screen "HAND_3" 800x480
   Button "Button_2" at 5,415 size 191x62; TextOff 'BACK'
      on Click: ActivateScreen("HAND_2", 0)
   TextField "Text field_12" at 206,35 size 347x29; Text 'CONVEYOR -1 START/STOP'
   Button "Button_21" at 690,7 size 11x44; TextOff 'Text'; PictureOff "Untitled_2"
   Button "Button_22" at 703,7 size 65x94; TextOff 'Text'; PictureOn "RIGHT_ARROW_ACTIVE"; PictureOff "RIGHT_ARROW_1"
      on Press: function_b14e0dd5("CONVEYOR -1 RUN FROM HMI", 0)
   TextField "Text field_13" at 623,7 size 64x44; Text 'START'
   TextField "Text field_18" at 623,57 size 64x44; Text 'Q1.0'
      Appearance <- "Tag_12"
   Button "Button_23" at 690,57 size 11x44; TextOff 'Text'; PictureOff "Untitled_2"
   Button "Button_24" at 33,7 size 65x94; TextOff 'Text'; PictureOn "LEFT_ARROW_ACTIVE"; PictureOff "LEFT_ARR"
      on Press: function_b14e0dd5("CONVEYOR -1 STOP FROM HMI", 0)
   TextField "Text field_19" at 119,7 size 64x44; Text 'STOP'
   Button "Button_25" at 101,7 size 11x44; TextOff 'Text'; PictureOff "Untitled_2"
   TextField "Text field_20" at 119,57 size 64x44; Text 'Q1.0'
      Appearance <- "Tag_12"
   Button "Button_26" at 101,57 size 11x44; TextOff 'Text'; PictureOff "Untitled_2"
   TextField "Text field_5" at 207,134 size 347x29; Text 'CONVEYOR -2 START/STOP'
   Button "Button_3" at 691,106 size 11x44; TextOff 'Text'; PictureOff "Untitled_2"
   Button "Button_4" at 704,106 size 65x94; TextOff 'Text'; PictureOn "RIGHT_ARROW_ACTIVE"; PictureOff "RIGHT_ARROW_1"
      on Press: function_b14e0dd5("CONVEYOR 2 RUN FROM HMI", 0)
   TextField "Text field_6" at 624,106 size 64x44; Text 'START'
   TextField "Text field_7" at 624,156 size 64x44; Text 'Q1.1'
      Appearance <- "Tag_13"
   Button "Button_5" at 691,156 size 11x44; TextOff 'Text'; PictureOff "Untitled_2"
   Button "Button_6" at 34,106 size 65x94; TextOff 'Text'; PictureOn "LEFT_ARROW_ACTIVE"; PictureOff "LEFT_ARR"
      on Press: function_b14e0dd5("CONVEYOR -2 STOP FROM HMI", 0)
   TextField "Text field_8" at 120,106 size 64x44; Text 'STOP'
   Button "Button_7" at 102,106 size 11x44; TextOff 'Text'; PictureOff "Untitled_2"
   TextField "Text field_9" at 120,156 size 64x44; Text 'Q1.1'
      Appearance <- "Tag_13"
   Button "Button_8" at 102,156 size 11x44; TextOff 'Text'; PictureOff "Untitled_2"
   TextField "Text field_1" at 236,241 size 327x29; Text 'PLUG HOLDER HOLD/UNHOLD'
   Button "Button_9" at 690,213 size 11x44; TextOff 'Text'; PictureOff "Untitled_2"
   Button "Button_10" at 703,213 size 65x94; TextOff 'Text'; PictureOn "RIGHT_ARROW_ACTIVE"; PictureOff "RIGHT_ARROW_1"
      on Press: function_b14e0dd5("HMI_GRIPPER_HOLD", 0)
      Appearance <- "HMI_GRIPPER_HOLD"
   TextField "Text field_2" at 623,213 size 64x44; Text 'HOLD'
      Appearance <- "GRIPPER_HOLD"
   TextField "Text field_3" at 623,263 size 64x44; Text 'Q6.2'
      Appearance <- "GRIPPER_HOLD"
   Button "Button_11" at 690,263 size 11x44; TextOff 'Text'; PictureOff "Untitled_2"
   Button "Button_12" at 33,213 size 65x94; TextOff 'Text'; PictureOn "LEFT_ARROW_ACTIVE"; PictureOff "LEFT_ARR"
      on Press: function_b14e0dd5("HMI_GRIPPER_UNHOLD", 0)
      Appearance <- "HMI_GRIPPER_UNHOLD"
   TextField "Text field_4" at 119,213 size 64x44; Text 'UNHOLD'
      Appearance <- "GRIPPER_UNHOLD"
   Button "Button_13" at 101,213 size 11x44; TextOff 'Text'; PictureOff "Untitled_2"
   TextField "Text field_10" at 119,263 size 64x44; Text 'Q6.3'
      Appearance <- "GRIPPER_UNHOLD"
   Button "Button_14" at 101,263 size 11x44; TextOff 'Text'; PictureOff "Untitled_2"
   Button "Button_27" at 609,416 size 191x63; TextOff 'HOME'
      on Click: ActivateScreen("MAIN", 0)
   Softkey "Softkey_F1" at 0,0 size 0x0
      on KeyDown: ActivateScreen("HAND_2", 0)
   Softkey "Softkey_F8" at 0,0 size 0x0
      on KeyDown: ActivateScreen("MAIN", 0)

screen "INPUT LIST" 800x480
   SymbolicIOField "Symbolic I/O field_1" at 160,52 size 153x48; TextOn '1'; TextOff '0'; TextList "INPUT ADDRESS"
      ProcessValue <- "0_BIT"
   SymbolicIOField "Symbolic I/O field_2" at 315,52 size 474x48; TextOn '1'; TextOff '0'; TextList "INPUT ADDRESS COMMENT"
      ProcessValue <- "0_BIT"
   TextField "Text field_1" at 36,14 size 71x23; Text 'STATUS'
   TextField "Text field_2" at 188,13 size 68x23; Text 'INPUTS'
   TextField "Text field_3" at 350,13 size 99x23; Text 'COMMENTS'
   SymbolicIOField "Symbolic I/O field_3" at 620,3 size 167x48; TextOn '1'; TextOff '0'; TextList "INPUT BYTE SELECTION"
      on Activate: function_dbe01993("0_BIT", 8, "BYTE SELECTION", 0); function_dbe01993("1_BIT", 8, "BYTE SELECTION", 1); function_dbe01993("2_BIT", 8, "BYTE SELECTION", 2); function_dbe01993("3_BIT", 8, "BYTE SELECTION", 3); function_dbe01993("4_BIT", 8, "BYTE SELECTION", 4); function_dbe01993("5_BIT", 8, "BYTE SELECTION", 5); function_dbe01993("6_BIT", 8, "BYTE SELECTION", 6); function_dbe01993("7_BIT", 8, "BYTE SELECTION", 7)
      on Change: function_dbe01993("0_BIT", 8, "BYTE SELECTION", 0); function_dbe01993("1_BIT", 8, "BYTE SELECTION", 1); function_dbe01993("2_BIT", 8, "BYTE SELECTION", 2); function_dbe01993("3_BIT", 8, "BYTE SELECTION", 3); function_dbe01993("4_BIT", 8, "BYTE SELECTION", 4); function_dbe01993("5_BIT", 8, "BYTE SELECTION", 5); function_dbe01993("6_BIT", 8, "BYTE SELECTION", 6); function_dbe01993("7_BIT", 8, "BYTE SELECTION", 7)
      ProcessValue <- "BYTE SELECTION"
   SymbolicIOField "Symbolic I/O field_4" at 160,102 size 153x48; TextOn '1'; TextOff '0'; TextList "INPUT ADDRESS"
      ProcessValue <- "1_BIT"
   SymbolicIOField "Symbolic I/O field_5" at 315,102 size 474x48; TextOn '1'; TextOff '0'; TextList "INPUT ADDRESS COMMENT"
      ProcessValue <- "1_BIT"
   Ellipse "Ellipse_2" at 31,103 size 89x46
      Appearance <- "I BIT_1"
   SymbolicIOField "Symbolic I/O field_6" at 160,151 size 153x48; TextOn '1'; TextOff '0'; TextList "INPUT ADDRESS"
      ProcessValue <- "2_BIT"
   SymbolicIOField "Symbolic I/O field_7" at 315,151 size 474x48; TextOn '1'; TextOff '0'; TextList "INPUT ADDRESS COMMENT"
      ProcessValue <- "2_BIT"
   Ellipse "Ellipse_3" at 31,152 size 89x46
      Appearance <- "I BIT_2"
   SymbolicIOField "Symbolic I/O field_8" at 162,200 size 153x48; TextOn '1'; TextOff '0'; TextList "INPUT ADDRESS"
      ProcessValue <- "3_BIT"
   SymbolicIOField "Symbolic I/O field_9" at 317,200 size 474x48; TextOn '1'; TextOff '0'; TextList "INPUT ADDRESS COMMENT"
      ProcessValue <- "3_BIT"
   SymbolicIOField "Symbolic I/O field_10" at 161,249 size 153x48; TextOn '1'; TextOff '0'; TextList "INPUT ADDRESS"
      ProcessValue <- "4_BIT"
   SymbolicIOField "Symbolic I/O field_11" at 316,249 size 474x48; TextOn '1'; TextOff '0'; TextList "INPUT ADDRESS COMMENT"
      ProcessValue <- "4_BIT"
   SymbolicIOField "Symbolic I/O field_12" at 162,298 size 153x48; TextOn '1'; TextOff '0'; TextList "INPUT ADDRESS"
      ProcessValue <- "5_BIT"
   SymbolicIOField "Symbolic I/O field_13" at 317,298 size 474x48; TextOn '1'; TextOff '0'; TextList "INPUT ADDRESS COMMENT"
      ProcessValue <- "5_BIT"
   SymbolicIOField "Symbolic I/O field_14" at 162,347 size 153x48; TextOn '1'; TextOff '0'; TextList "INPUT ADDRESS"
      ProcessValue <- "6_BIT"
   SymbolicIOField "Symbolic I/O field_15" at 317,347 size 474x48; TextOn '1'; TextOff '0'; TextList "INPUT ADDRESS COMMENT"
      ProcessValue <- "6_BIT"
   SymbolicIOField "Symbolic I/O field_16" at 163,396 size 153x48; TextOn '1'; TextOff '0'; TextList "INPUT ADDRESS"
      ProcessValue <- "7_BIT"
   SymbolicIOField "Symbolic I/O field_17" at 317,395 size 474x48; TextOn '1'; TextOff '0'; TextList "INPUT ADDRESS COMMENT"
      ProcessValue <- "7_BIT"
   Ellipse "Ellipse_4" at 31,201 size 89x46
      Appearance <- "I BIT_3"
   Ellipse "Ellipse_5" at 31,249 size 89x46
      Appearance <- "I BIT_4"
   Ellipse "Ellipse_6" at 31,300 size 89x46
      Appearance <- "I BIT_5"
   Ellipse "Ellipse_7" at 31,347 size 89x46
      Appearance <- "I BIT_6"
   Ellipse "Ellipse_8" at 31,396 size 89x46
      Appearance <- "I BIT_7"
   Ellipse "Ellipse_1" at 31,53 size 89x46
      Appearance <- "I BIT_0"
   Button "Button_2" at 599,442 size 191x35; TextOff 'HOME'
      on Click: ActivateScreen("MAIN", 0)
   Softkey "Softkey_F8" at 0,0 size 0x0
      on KeyDown: ActivateScreen("MAIN", 0)

screen "OUTPUT LIST" 800x480
   SymbolicIOField "Symbolic I/O field_1" at 160,52 size 153x48; TextOn '1'; TextOff '0'; TextList "OUTPUT ADDRESS"
      ProcessValue <- "0_BIT"
   SymbolicIOField "Symbolic I/O field_2" at 315,52 size 474x48; TextOn '1'; TextOff '0'; TextList "OUTADDRESS COMMENT"
      ProcessValue <- "0_BIT"
   TextField "Text field_1" at 36,14 size 71x23; Text 'STATUS'
   TextField "Text field_2" at 188,13 size 68x23; Text 'INPUTS'
   TextField "Text field_3" at 350,13 size 99x23; Text 'COMMENTS'
   SymbolicIOField "Symbolic I/O field_3" at 620,3 size 167x48; TextOn '1'; TextOff '0'; TextList "OUT BYTE SELECTION"
      on Activate: function_dbe01993("0_BIT", 8, "BYTE SELECTION", 0); function_dbe01993("1_BIT", 8, "BYTE SELECTION", 1); function_dbe01993("2_BIT", 8, "BYTE SELECTION", 2); function_dbe01993("3_BIT", 8, "BYTE SELECTION", 3); function_dbe01993("4_BIT", 8, "BYTE SELECTION", 4); function_dbe01993("5_BIT", 8, "BYTE SELECTION", 5); function_dbe01993("6_BIT", 8, "BYTE SELECTION", 6); function_dbe01993("7_BIT", 8, "BYTE SELECTION", 7)
      on Change: function_dbe01993("0_BIT", 8, "BYTE SELECTION", 0); function_dbe01993("1_BIT", 8, "BYTE SELECTION", 1); function_dbe01993("2_BIT", 8, "BYTE SELECTION", 2); function_dbe01993("3_BIT", 8, "BYTE SELECTION", 3); function_dbe01993("4_BIT", 8, "BYTE SELECTION", 4); function_dbe01993("5_BIT", 8, "BYTE SELECTION", 5); function_dbe01993("6_BIT", 8, "BYTE SELECTION", 6); function_dbe01993("7_BIT", 8, "BYTE SELECTION", 7)
      ProcessValue <- "BYTE SELECTION"
   SymbolicIOField "Symbolic I/O field_4" at 160,102 size 153x48; TextOn '1'; TextOff '0'; TextList "OUTPUT ADDRESS"
      ProcessValue <- "1_BIT"
   SymbolicIOField "Symbolic I/O field_5" at 315,102 size 474x48; TextOn '1'; TextOff '0'; TextList "OUTADDRESS COMMENT"
      ProcessValue <- "1_BIT"
   Ellipse "Ellipse_2" at 31,103 size 89x46
      Appearance <- "Q BIT_1"
   SymbolicIOField "Symbolic I/O field_6" at 160,151 size 153x48; TextOn '1'; TextOff '0'; TextList "OUTPUT ADDRESS"
      ProcessValue <- "2_BIT"
   SymbolicIOField "Symbolic I/O field_7" at 315,151 size 474x48; TextOn '1'; TextOff '0'; TextList "OUTADDRESS COMMENT"
      ProcessValue <- "2_BIT"
   Ellipse "Ellipse_3" at 31,152 size 89x46
      Appearance <- "Q BIT_2"
   SymbolicIOField "Symbolic I/O field_8" at 162,200 size 153x48; TextOn '1'; TextOff '0'; TextList "OUTPUT ADDRESS"
      ProcessValue <- "3_BIT"
   SymbolicIOField "Symbolic I/O field_9" at 317,200 size 474x48; TextOn '1'; TextOff '0'; TextList "OUTADDRESS COMMENT"
      ProcessValue <- "3_BIT"
   SymbolicIOField "Symbolic I/O field_10" at 161,249 size 153x48; TextOn '1'; TextOff '0'; TextList "OUTPUT ADDRESS"
      ProcessValue <- "4_BIT"
   SymbolicIOField "Symbolic I/O field_11" at 316,249 size 474x48; TextOn '1'; TextOff '0'; TextList "OUTADDRESS COMMENT"
      ProcessValue <- "4_BIT"
   SymbolicIOField "Symbolic I/O field_12" at 162,298 size 153x48; TextOn '1'; TextOff '0'; TextList "OUTPUT ADDRESS"
      ProcessValue <- "5_BIT"
   SymbolicIOField "Symbolic I/O field_13" at 317,298 size 474x48; TextOn '1'; TextOff '0'; TextList "OUTADDRESS COMMENT"
      ProcessValue <- "5_BIT"
   SymbolicIOField "Symbolic I/O field_14" at 162,347 size 153x48; TextOn '1'; TextOff '0'; TextList "OUTPUT ADDRESS"
      ProcessValue <- "6_BIT"
   SymbolicIOField "Symbolic I/O field_15" at 317,347 size 474x48; TextOn '1'; TextOff '0'; TextList "OUTADDRESS COMMENT"
      ProcessValue <- "6_BIT"
   SymbolicIOField "Symbolic I/O field_16" at 163,396 size 153x48; TextOn '1'; TextOff '0'; TextList "OUTPUT ADDRESS"
      ProcessValue <- "7_BIT"
   SymbolicIOField "Symbolic I/O field_17" at 317,395 size 474x48; TextOn '1'; TextOff '0'; TextList "OUTADDRESS COMMENT"
      ProcessValue <- "7_BIT"
   Ellipse "Ellipse_4" at 31,201 size 89x46
      Appearance <- "Q BIT_3"
   Ellipse "Ellipse_5" at 31,249 size 89x46
      Appearance <- "Q BIT_4"
   Ellipse "Ellipse_6" at 31,300 size 89x46
      Appearance <- "Q BIT_5"
   Ellipse "Ellipse_7" at 31,347 size 89x46
      Appearance <- "Q BIT_6"
   Ellipse "Ellipse_8" at 31,396 size 89x46
      Appearance <- "Q BIT_7"
   Ellipse "Ellipse_1" at 31,53 size 89x46
      Appearance <- "Q BIT_0"
   Button "Button_2" at 599,436 size 191x41; TextOff 'HOME'
      on Click: ActivateScreen("MAIN", 0)
   Softkey "Softkey_F8" at 0,0 size 0x0
      on KeyDown: ActivateScreen("MAIN", 0)

screen "ALARMS" 800x480
   Softkey "[!Invalid!]Softkey_#mig1" at -133,-132 size 72x51
      on PressedNotHandled: ActivateScreen("MAIN", 0)
   Softkey "[!Invalid!]Softkey_#mig2" at -133,-132 size 72x51
      on KeyDown: ActivateScreen("MAIN", 0)
   Softkey "Softkey_F1" at 14,429 size 72x51
      on KeyDown: ActivateScreen("HAND_1", 0)
   AlarmView "P_MESSAGE_VIEW_1" at 0,0 size 791x426; ColumnTextDevice 'PLC / API / ПЛК'; ColumnTextAckGroup 'GR / Gruppe quittieren / Acusar grupo / Acquitter le groupe / Conferma gruppo / 确认组 / ｸﾞﾙｰﾌﾟを確認 / Квитировать группу'; ColumnTextAlarmState 'Status / Estado / Etat / Stato / 状态 / ｽﾃｰﾀｽ / Статус'; ColumnTextAlarmText 'MessageViewAlarms / Text / Texto / Texte / Testo / 文本 / ﾃｷｽﾄ / Текст'; ColumnTextTime 'Time / Zeit / Hora / Heure / Tempo / 时间 / 時間 / Время'; ColumnTextDate 'Date / Datum / Fecha / Data / 日期 / 日付 / Дата'; ColumnTextNumber 'No. / Nr. / N.º. / N°. / 编号. / 番号 / №'
   Button "Button_3" at 3,426 size 97x53; TextOff 'HAND'
      on Click: ActivateScreen("HAND_1", 0)
   Button "Button_1" at 694,426 size 97x53; TextOff 'MAIN'
      on Click: ActivateScreen("MAIN", 0)
   Softkey "Softkey_F8" at 714,429 size 72x51
      on KeyDown: ActivateScreen("MAIN", 0)

screen "MAIN" 800x480
   Softkey "Softkey_F1" at 14,429 size 72x51
      on KeyDown: ActivateScreen("ALARMS", 0)
   Softkey "[!Invalid!]Softkey_#mig2" at -133,-132 size 72x51
      on PressedNotHandled: function_efd93a16()
   Softkey "[!Invalid!]Softkey_#mig4" at -133,-132 size 72x51
      on KeyDown: ActivateScreen("MAIN", 0)
   Softkey "[!Invalid!]Softkey_#mig5" at -133,-132 size 72x51
      on KeyDown: ActivateScreen("AUI", 0)
   Softkey "[!Invalid!]Softkey_#mig6" at -133,-132 size 72x51
      on KeyDown: function_b14e0dd5("#mig1#RESET_COUNT", 0)
   Softkey "Softkey_F4" at 314,429 size 72x51
      on KeyDown: ActivateScreen("HAND_1", 0)
   Softkey "Softkey_F5" at 414,429 size 72x51
      on KeyUp: ActivateScreen("INPUT LIST", 0)
   GraphicView "Graphic view_1" at 7,2 size 189x56; Picture "BOSCH"
   TextField "Text Field_6" at 212,3 size 452x55; Text 'AUTO-5 UNLOADING'
   TextField "Text field_2" at 542,131 size 236x43; Text 'PLUGS COUNT'
   Button "Button_3" at 7,413 size 97x63; TextOff 'ALARM'
      on Click: ActivateScreen("ALARMS", 0)
   IOField "MAIN_2_1" at 574,194 size 165x84; FormatPattern 9999
      ProcessValue <- "RETENTIVES_PLUG COUNTER"
   Button "Button_1" at 295,414 size 97x62; TextOff 'HAND'
      on Click: ActivateScreen("HAND_1", 0)
   Button "Button_12" at 542,415 size 138x61; TextOff 'OUTPUT LIST'
      on Click: ActivateScreen("OUTPUT LIST", 0)
   TextField "Text field_1" at 216,75 size 368x38; Text 'ALL UNIT INITIAL SCREEN'
   DateTimeField "Date/time field_1" at 680,3 size 111x32
   DateTimeField "Date/time field_2" at 680,40 size 110x31
   TextField "Text field_4" at 29,145 size 386x29; Text 'PLUG SENSOR MOUNTED ON CHUTE'
   Circle "Circle_63" at 486,146 size 28x28
      Appearance <- "PLUG SENSOR MOUNTED ON CHUTE_INPUT"
   TextField "Text field_5" at 25,190 size 390x29; Text 'PLUG LIFTING CYLINDER FORWARD'
   TextField "Text field_3" at 57,232 size 356x29; Text 'TRAY LIFTING HEIGHT DOWN RS'
   TextField "Text field_7" at 28,319 size 390x29; Text 'TRAY LIFTING DOWN READ SWITCH'
   TextField "Text field_8" at 66,277 size 352x29; Text 'PLUG LIFTING UP READ SWITCH'
   TextField "Text field_10" at 423,145 size 48x29; Text 'I1.0'
   TextField "Text field_9" at 423,189 size 48x29; Text 'I3.5'
   TextField "Text field_11" at 423,233 size 48x29; Text 'I2.6'
   TextField "Text field_12" at 423,277 size 48x29; Text 'I3.0'
   TextField "Text field_13" at 423,321 size 48x29; Text 'I3.4'
   Circle "Circle_1" at 486,190 size 28x28
      Appearance <- "PLUG LIFTING CYLINDER_FORWARD"
   Circle "Circle_2" at 486,234 size 28x28
      Appearance <- "TRAY LIFTING HEIGHT LEVELING_DOWN"
   Circle "Circle_3" at 486,278 size 28x28
      Appearance <- "TRAY LIFTING CYLINDER _DOWN"
   Circle "Circle_4" at 486,322 size 28x28
      Appearance <- "PLUG LIFTING CYLINDER_UP"
   Button "Button_2" at 399,415 size 134x63; TextOff 'INPUT LIST'
      on Click: ActivateScreen("INPUT LIST", 0)
   TextField "Text field_14" at 187,365 size 229x34; Text 'ALL UNIT INITIAL'
   TextField "Text field_15" at 419,367 size 54x29; Text 'Q0.2'
   Circle "Circle_5" at 486,365 size 29x29
      Appearance <- "ALL_UNIT_INITIAL"
   TextField "Text field_16" at 523,314 size 142x22; Text 'INITIAL RESET PB'
   TextField "Text field_17" at 552,319 size 14x25; Text 'Text'
   TextField "Text field_18" at 529,362 size 129x22; Text 'FAULT RESET PB'
   TextField "Text field_19" at 584,331 size 25x34; Text '+'
   TextField "Text field_20" at 691,329 size 104x22; Text 'PLUG COUNT'
   TextField "Text field_21" at 715,355 size 53x22; Text 'RESET'
   TextField "Text field_22" at 667,340 size 25x34; Text '='
   Button "Button_4" at 687,415 size 105x62; TextOff 'TRAY INITIAL'
      on Click: ActivateScreen("HAND_1", 0)
   Softkey "Softkey_F8" at 714,429 size 72x51
      on KeyDown: function_b14e0dd5("HMI_TRAY_PRESENT_INITIAL", 0)
      on KeyUp: ResetBit("HMI_TRAY_PRESENT_INITIAL")
   Softkey "Softkey_F7" at 0,0 size 0x0
      on KeyUp: ActivateScreen("OUTPUT LIST", 0)
*)